// TIA Portal V15.1 export
// export: Created 2024-05-17T05:38:59.5834556Z, ExportSetting WithDefaults, DisplayName Totally Integrated Automation Portal, DisplayVersion V15.1 Update 5, DisplayName TIA Portal Openness, DisplayVersion V15.1 Update 5, DisplayName SINAMICS Startdrive Advanced, DisplayVersion V15.1, DisplayName G130, G150, S120, S150, SINAMICS MV, S210, DisplayVersion V15.1, DisplayName G110M, G120, G120C, G120D, G120P, DisplayVersion V15.1, DisplayName STEP 7 Professional, DisplayVersion V15.1 Update 5, DisplayName STEP 7 Safety, DisplayVersion V15.1, DisplayName WinCC Professional, DisplayVersion V15.1 Update 5, DisplayName SIMATIC Visualization Architect, DisplayVersion V15.1
FUNCTION "209000NCP01PNIODiag" : Void   // FC270, FBD
TITLE = 209000NCP01PNIODiag
{ S7_Optimized_Access := 'FALSE' }
AUTHOR : JS
NAME : Mot001
VERSION : 0.1
// stored: AutoNumber false, IsIECCheckEnabled false, SetENOAutomatically False, UDAEnableTagReadback false
   VAR_OUTPUT
      O_AlarmA : Bool;   // Alarm A
      O_AlarmB : Bool;   // Alarm B
      O_AlarmC : Bool;   // Alarm C
      O_AlarmD : Bool;   // Alarm D
      O_AlarmABCondition : Bool;   // Alarms resetable
      H_IAnim : Word;   // Animation bits to Icon in WinCC
   END_VAR
   VAR_TEMP   // added for the SCL form of the ladder/FBD networks
      _w1 : Bool;
   END_VAR
BEGIN

REGION Network 1: **** 1 - Inputs **** HMI Cmd
   // Extract HMI Cmd
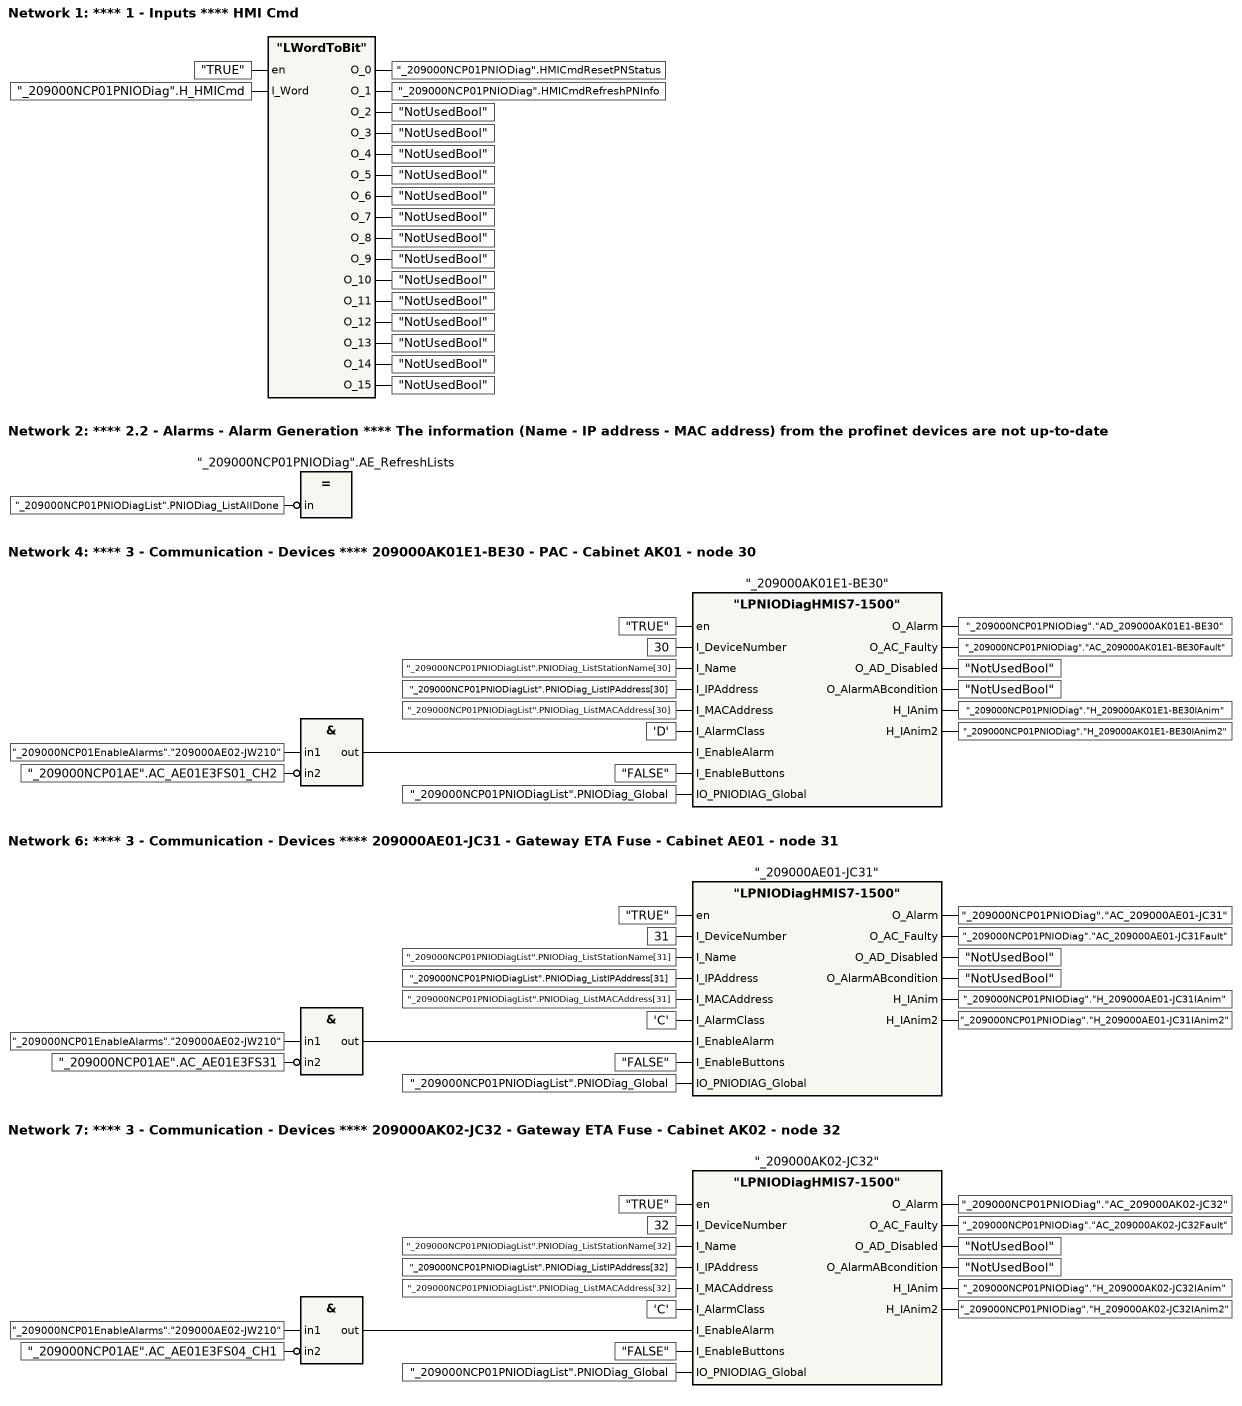
   IF "TRUE" THEN
       "LWordToBit"(I_Word := "_209000NCP01PNIODiag".H_HMICmd,
                    O_0 => "_209000NCP01PNIODiag".HMICmdResetPNStatus,
                    O_1 => "_209000NCP01PNIODiag".HMICmdRefreshPNInfo,
                    O_2 => "NotUsedBool",
                    O_3 => "NotUsedBool",
                    O_4 => "NotUsedBool",
                    O_5 => "NotUsedBool",
                    O_6 => "NotUsedBool",
                    O_7 => "NotUsedBool",
                    O_8 => "NotUsedBool",
                    O_9 => "NotUsedBool",
                    O_10 => "NotUsedBool",
                    O_11 => "NotUsedBool",
                    O_12 => "NotUsedBool",
                    O_13 => "NotUsedBool",
                    O_14 => "NotUsedBool",
                    O_15 => "NotUsedBool");
   END_IF;
END_REGION

REGION Network 2: **** 2.2 - Alarms - Alarm Generation **** The information (Name - IP address - MAC address) from the profinet devices are not up-to-date
   // The information (Name - IP address - MAC address) from the profinet devices are not up-to-date
   "_209000NCP01PNIODiag".AE_RefreshLists := NOT "_209000NCP01PNIODiagList".PNIODiag_ListAllDone;
END_REGION

REGION Network 3: **** --------------------- PAC --------------------- ****
END_REGION

REGION Network 4: **** 3 - Communication - Devices **** 209000AK01E1-BE30 - PAC - Cabinet AK01 - node 30
   // Profinet device don't exist - PAC - Cabinet AK01 - node 30
   IF "TRUE" THEN
       "_209000AK01E1-BE30"(I_DeviceNumber := 30,   // "LPNIODiagHMIS7-1500"
                            I_Name := "_209000NCP01PNIODiagList".PNIODiag_ListStationName[30],
                            I_IPAddress := "_209000NCP01PNIODiagList".PNIODiag_ListIPAddress[30],
                            I_MACAddress := "_209000NCP01PNIODiagList".PNIODiag_ListMACAddress[30],
                            I_AlarmClass := 'D',
                            I_EnableAlarm := "_209000NCP01EnableAlarms"."209000AE02-JW210" AND NOT "_209000NCP01AE".AC_AE01E3FS01_CH2,
                            I_EnableButtons := "FALSE",
                            IO_PNIODIAG_Global := "_209000NCP01PNIODiagList".PNIODiag_Global,
                            O_Alarm => "_209000NCP01PNIODiag"."AD_209000AK01E1-BE30",
                            O_AC_Faulty => "_209000NCP01PNIODiag"."AC_209000AK01E1-BE30Fault",
                            O_AD_Disabled => "NotUsedBool",
                            O_AlarmABcondition => "NotUsedBool",
                            H_IAnim => "_209000NCP01PNIODiag"."H_209000AK01E1-BE30IAnim",
                            H_IAnim2 => "_209000NCP01PNIODiag"."H_209000AK01E1-BE30IAnim2");
   END_IF;
END_REGION

REGION Network 5: **** --------------------- Gateway --------------------- ****
END_REGION

REGION Network 6: **** 3 - Communication - Devices **** 209000AE01-JC31 - Gateway ETA Fuse - Cabinet AE01 - node 31
   // Profinet device don't exist - Gateway ETA Fuse - Cabinet AE01 - node 31
   IF "TRUE" THEN
       "_209000AE01-JC31"(I_DeviceNumber := 31,   // "LPNIODiagHMIS7-1500"
                          I_Name := "_209000NCP01PNIODiagList".PNIODiag_ListStationName[31],
                          I_IPAddress := "_209000NCP01PNIODiagList".PNIODiag_ListIPAddress[31],
                          I_MACAddress := "_209000NCP01PNIODiagList".PNIODiag_ListMACAddress[31],
                          I_AlarmClass := 'C',
                          I_EnableAlarm := "_209000NCP01EnableAlarms"."209000AE02-JW210" AND NOT "_209000NCP01AE".AC_AE01E3FS31,
                          I_EnableButtons := "FALSE",
                          IO_PNIODIAG_Global := "_209000NCP01PNIODiagList".PNIODiag_Global,
                          O_Alarm => "_209000NCP01PNIODiag"."AC_209000AE01-JC31",
                          O_AC_Faulty => "_209000NCP01PNIODiag"."AC_209000AE01-JC31Fault",
                          O_AD_Disabled => "NotUsedBool",
                          O_AlarmABcondition => "NotUsedBool",
                          H_IAnim => "_209000NCP01PNIODiag"."H_209000AE01-JC31IAnim",
                          H_IAnim2 => "_209000NCP01PNIODiag"."H_209000AE01-JC31IAnim2");
   END_IF;
END_REGION

REGION Network 7: **** 3 - Communication - Devices **** 209000AK02-JC32 - Gateway ETA Fuse - Cabinet AK02 - node 32
   // Profinet device don't exist - Gateway ETA Fuse - Cabinet AK02 - node 32
   IF "TRUE" THEN
       "_209000AK02-JC32"(I_DeviceNumber := 32,   // "LPNIODiagHMIS7-1500"
                          I_Name := "_209000NCP01PNIODiagList".PNIODiag_ListStationName[32],
                          I_IPAddress := "_209000NCP01PNIODiagList".PNIODiag_ListIPAddress[32],
                          I_MACAddress := "_209000NCP01PNIODiagList".PNIODiag_ListMACAddress[32],
                          I_AlarmClass := 'C',
                          I_EnableAlarm := "_209000NCP01EnableAlarms"."209000AE02-JW210" AND NOT "_209000NCP01AE".AC_AE01E3FS04_CH1,
                          I_EnableButtons := "FALSE",
                          IO_PNIODIAG_Global := "_209000NCP01PNIODiagList".PNIODiag_Global,
                          O_Alarm => "_209000NCP01PNIODiag"."AC_209000AK02-JC32",
                          O_AC_Faulty => "_209000NCP01PNIODiag"."AC_209000AK02-JC32Fault",
                          O_AD_Disabled => "NotUsedBool",
                          O_AlarmABcondition => "NotUsedBool",
                          H_IAnim => "_209000NCP01PNIODiag"."H_209000AK02-JC32IAnim",
                          H_IAnim2 => "_209000NCP01PNIODiag"."H_209000AK02-JC32IAnim2");
   END_IF;
END_REGION

REGION Network 8: **** --------------------- ET200sp I/O --------------------- ****
END_REGION

REGION Network 9: **** 3 - Communication - Devices **** 209000AK01-JW35 - ET200sp I/O - Busnode AK01 - node 35
   // Profinet device don't exist - ET200sp I/O - Busnode AK01 - node 35
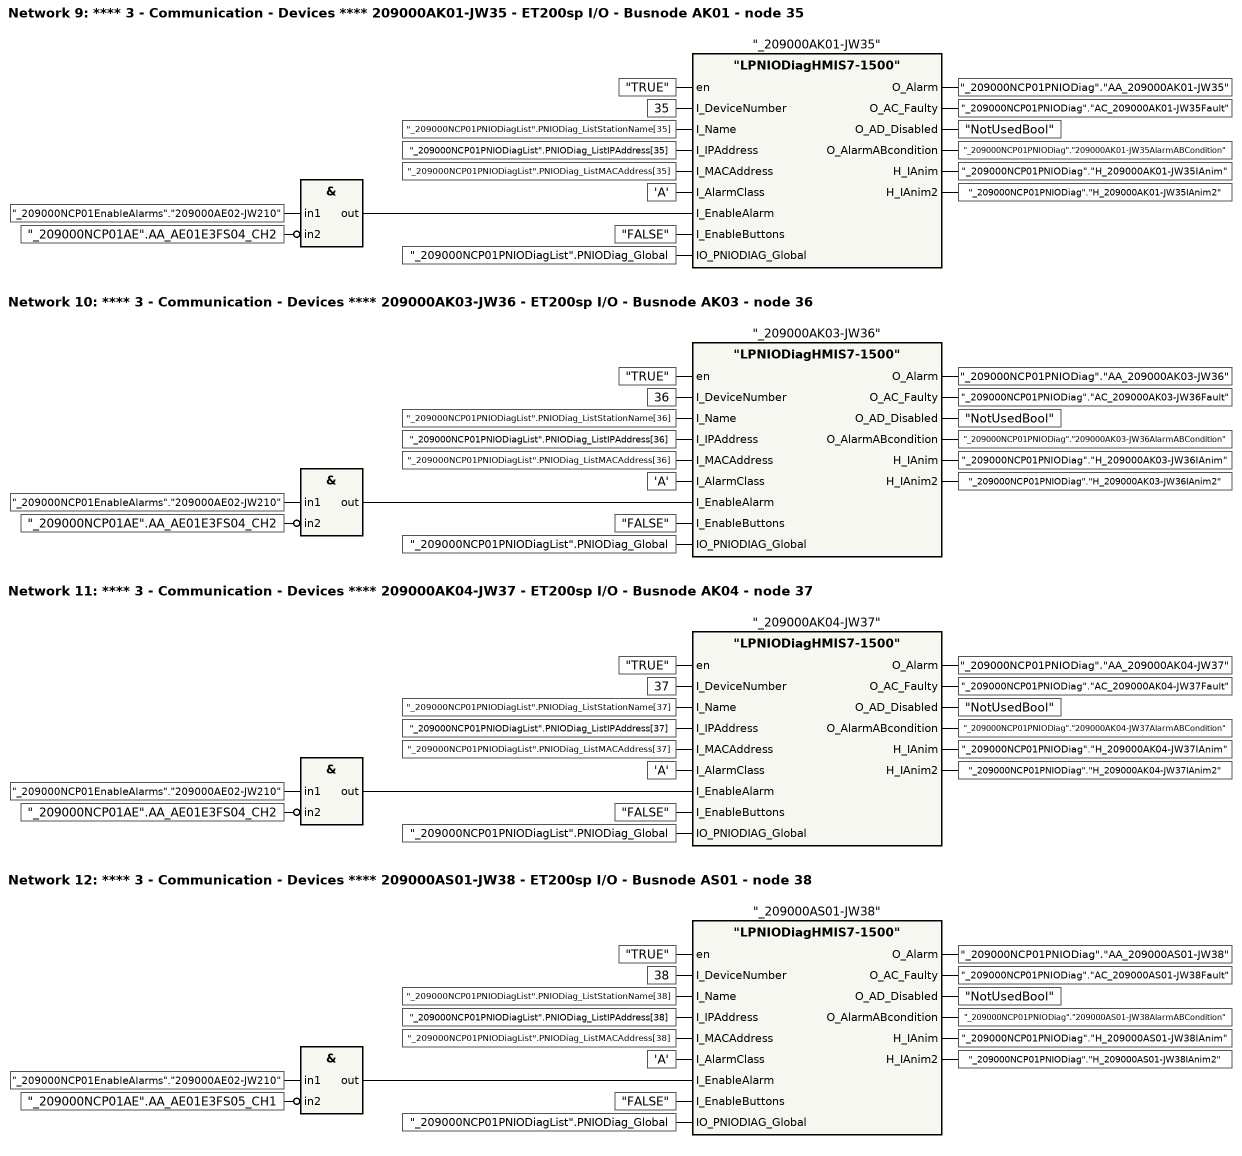
   IF "TRUE" THEN
       "_209000AK01-JW35"(I_DeviceNumber := 35,   // "LPNIODiagHMIS7-1500"
                          I_Name := "_209000NCP01PNIODiagList".PNIODiag_ListStationName[35],
                          I_IPAddress := "_209000NCP01PNIODiagList".PNIODiag_ListIPAddress[35],
                          I_MACAddress := "_209000NCP01PNIODiagList".PNIODiag_ListMACAddress[35],
                          I_AlarmClass := 'A',
                          I_EnableAlarm := "_209000NCP01EnableAlarms"."209000AE02-JW210" AND NOT "_209000NCP01AE".AA_AE01E3FS04_CH2,
                          I_EnableButtons := "FALSE",
                          IO_PNIODIAG_Global := "_209000NCP01PNIODiagList".PNIODiag_Global,
                          O_Alarm => "_209000NCP01PNIODiag"."AA_209000AK01-JW35",
                          O_AC_Faulty => "_209000NCP01PNIODiag"."AC_209000AK01-JW35Fault",
                          O_AD_Disabled => "NotUsedBool",
                          O_AlarmABcondition => "_209000NCP01PNIODiag"."209000AK01-JW35AlarmABCondition",
                          H_IAnim => "_209000NCP01PNIODiag"."H_209000AK01-JW35IAnim",
                          H_IAnim2 => "_209000NCP01PNIODiag"."H_209000AK01-JW35IAnim2");
   END_IF;
END_REGION

REGION Network 10: **** 3 - Communication - Devices **** 209000AK03-JW36 - ET200sp I/O - Busnode AK03 - node 36
   // Profinet device don't exist - ET200sp I/O - Busnode AK03 - node 36
   IF "TRUE" THEN
       "_209000AK03-JW36"(I_DeviceNumber := 36,   // "LPNIODiagHMIS7-1500"
                          I_Name := "_209000NCP01PNIODiagList".PNIODiag_ListStationName[36],
                          I_IPAddress := "_209000NCP01PNIODiagList".PNIODiag_ListIPAddress[36],
                          I_MACAddress := "_209000NCP01PNIODiagList".PNIODiag_ListMACAddress[36],
                          I_AlarmClass := 'A',
                          I_EnableAlarm := "_209000NCP01EnableAlarms"."209000AE02-JW210" AND NOT "_209000NCP01AE".AA_AE01E3FS04_CH2,
                          I_EnableButtons := "FALSE",
                          IO_PNIODIAG_Global := "_209000NCP01PNIODiagList".PNIODiag_Global,
                          O_Alarm => "_209000NCP01PNIODiag"."AA_209000AK03-JW36",
                          O_AC_Faulty => "_209000NCP01PNIODiag"."AC_209000AK03-JW36Fault",
                          O_AD_Disabled => "NotUsedBool",
                          O_AlarmABcondition => "_209000NCP01PNIODiag"."209000AK03-JW36AlarmABCondition",
                          H_IAnim => "_209000NCP01PNIODiag"."H_209000AK03-JW36IAnim",
                          H_IAnim2 => "_209000NCP01PNIODiag"."H_209000AK03-JW36IAnim2");
   END_IF;
END_REGION

REGION Network 11: **** 3 - Communication - Devices **** 209000AK04-JW37 - ET200sp I/O - Busnode AK04 - node 37
   // Profinet device don't exist - ET200sp I/O - Busnode AK04 - node 37
   IF "TRUE" THEN
       "_209000AK04-JW37"(I_DeviceNumber := 37,   // "LPNIODiagHMIS7-1500"
                          I_Name := "_209000NCP01PNIODiagList".PNIODiag_ListStationName[37],
                          I_IPAddress := "_209000NCP01PNIODiagList".PNIODiag_ListIPAddress[37],
                          I_MACAddress := "_209000NCP01PNIODiagList".PNIODiag_ListMACAddress[37],
                          I_AlarmClass := 'A',
                          I_EnableAlarm := "_209000NCP01EnableAlarms"."209000AE02-JW210" AND NOT "_209000NCP01AE".AA_AE01E3FS04_CH2,
                          I_EnableButtons := "FALSE",
                          IO_PNIODIAG_Global := "_209000NCP01PNIODiagList".PNIODiag_Global,
                          O_Alarm => "_209000NCP01PNIODiag"."AA_209000AK04-JW37",
                          O_AC_Faulty => "_209000NCP01PNIODiag"."AC_209000AK04-JW37Fault",
                          O_AD_Disabled => "NotUsedBool",
                          O_AlarmABcondition => "_209000NCP01PNIODiag"."209000AK04-JW37AlarmABCondition",
                          H_IAnim => "_209000NCP01PNIODiag"."H_209000AK04-JW37IAnim",
                          H_IAnim2 => "_209000NCP01PNIODiag"."H_209000AK04-JW37IAnim2");
   END_IF;
END_REGION

REGION Network 12: **** 3 - Communication - Devices **** 209000AS01-JW38 - ET200sp I/O - Busnode AS01 - node 38
   // Profinet device don't exist - ET200sp I/O - Busnode AS01 - node 38
   IF "TRUE" THEN
       "_209000AS01-JW38"(I_DeviceNumber := 38,   // "LPNIODiagHMIS7-1500"
                          I_Name := "_209000NCP01PNIODiagList".PNIODiag_ListStationName[38],
                          I_IPAddress := "_209000NCP01PNIODiagList".PNIODiag_ListIPAddress[38],
                          I_MACAddress := "_209000NCP01PNIODiagList".PNIODiag_ListMACAddress[38],
                          I_AlarmClass := 'A',
                          I_EnableAlarm := "_209000NCP01EnableAlarms"."209000AE02-JW210" AND NOT "_209000NCP01AE".AA_AE01E3FS05_CH1,
                          I_EnableButtons := "FALSE",
                          IO_PNIODIAG_Global := "_209000NCP01PNIODiagList".PNIODiag_Global,
                          O_Alarm => "_209000NCP01PNIODiag"."AA_209000AS01-JW38",
                          O_AC_Faulty => "_209000NCP01PNIODiag"."AC_209000AS01-JW38Fault",
                          O_AD_Disabled => "NotUsedBool",
                          O_AlarmABcondition => "_209000NCP01PNIODiag"."209000AS01-JW38AlarmABCondition",
                          H_IAnim => "_209000NCP01PNIODiag"."H_209000AS01-JW38IAnim",
                          H_IAnim2 => "_209000NCP01PNIODiag"."H_209000AS01-JW38IAnim2");
   END_IF;
END_REGION

REGION Network 13: **** 3 - Communication - Devices **** 209000AS02-JW39 - ET200sp I/O - Busnode AS02 - node 39
   // Profinet device don't exist - ET200sp I/O - Busnode AS02 - node 39
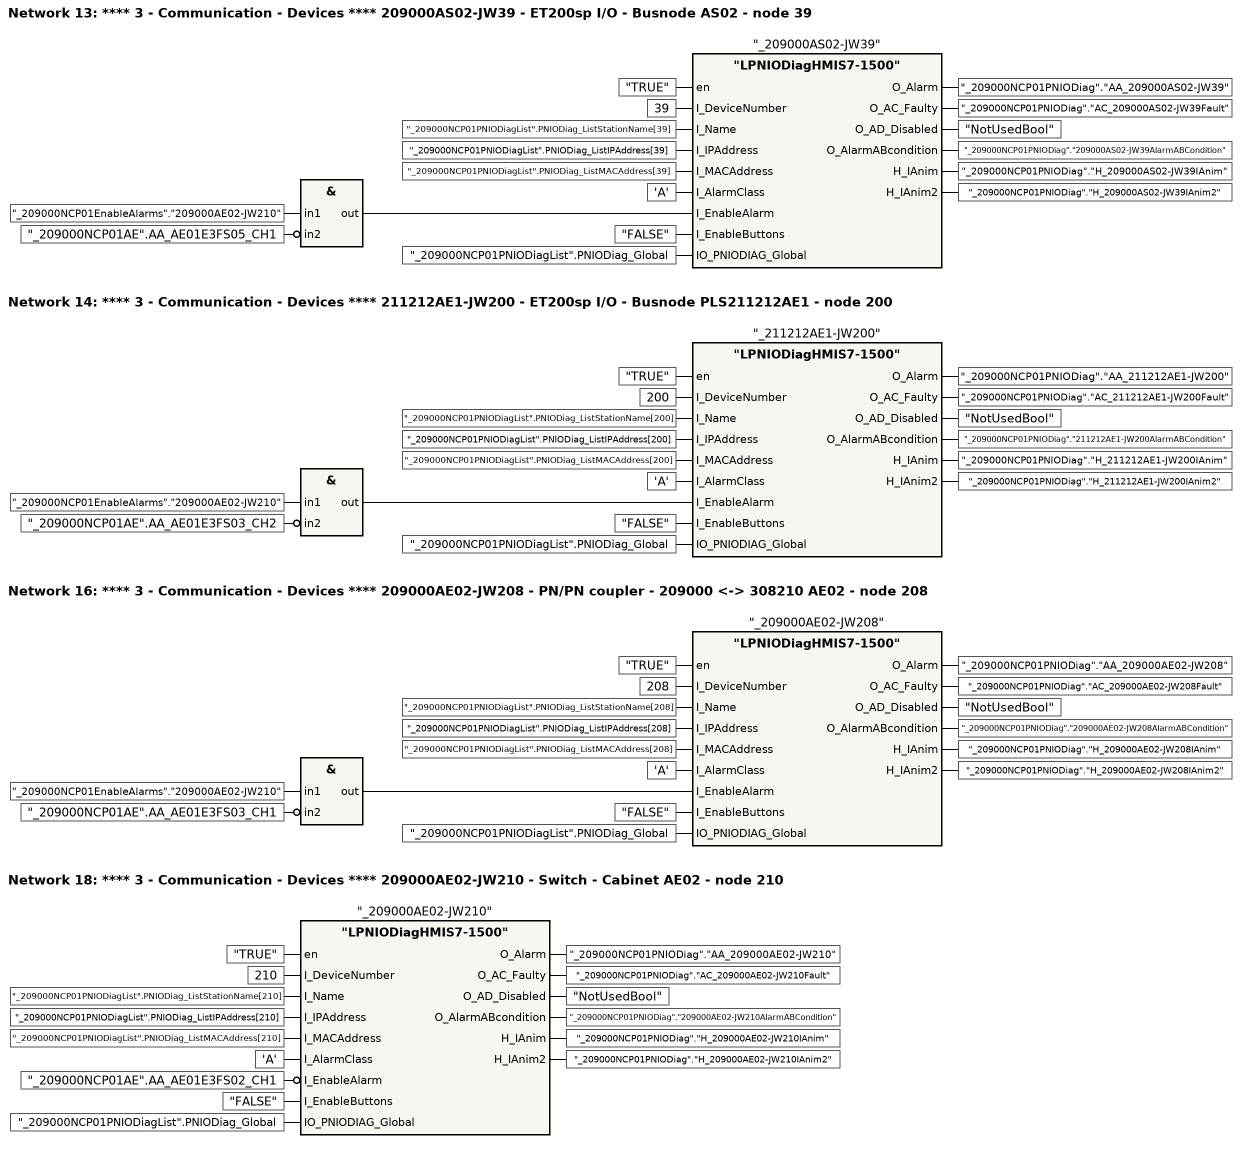
   IF "TRUE" THEN
       "_209000AS02-JW39"(I_DeviceNumber := 39,   // "LPNIODiagHMIS7-1500"
                          I_Name := "_209000NCP01PNIODiagList".PNIODiag_ListStationName[39],
                          I_IPAddress := "_209000NCP01PNIODiagList".PNIODiag_ListIPAddress[39],
                          I_MACAddress := "_209000NCP01PNIODiagList".PNIODiag_ListMACAddress[39],
                          I_AlarmClass := 'A',
                          I_EnableAlarm := "_209000NCP01EnableAlarms"."209000AE02-JW210" AND NOT "_209000NCP01AE".AA_AE01E3FS05_CH1,
                          I_EnableButtons := "FALSE",
                          IO_PNIODIAG_Global := "_209000NCP01PNIODiagList".PNIODiag_Global,
                          O_Alarm => "_209000NCP01PNIODiag"."AA_209000AS02-JW39",
                          O_AC_Faulty => "_209000NCP01PNIODiag"."AC_209000AS02-JW39Fault",
                          O_AD_Disabled => "NotUsedBool",
                          O_AlarmABcondition => "_209000NCP01PNIODiag"."209000AS02-JW39AlarmABCondition",
                          H_IAnim => "_209000NCP01PNIODiag"."H_209000AS02-JW39IAnim",
                          H_IAnim2 => "_209000NCP01PNIODiag"."H_209000AS02-JW39IAnim2");
   END_IF;
END_REGION

REGION Network 14: **** 3 - Communication - Devices **** 211212AE1-JW200 - ET200sp I/O - Busnode PLS211212AE1 - node 200
   // Profinet device don't exist - ET200sp I/O - Busnode PLS211212AE1 - node 200
   IF "TRUE" THEN
       "_211212AE1-JW200"(I_DeviceNumber := 200,   // "LPNIODiagHMIS7-1500"
                          I_Name := "_209000NCP01PNIODiagList".PNIODiag_ListStationName[200],
                          I_IPAddress := "_209000NCP01PNIODiagList".PNIODiag_ListIPAddress[200],
                          I_MACAddress := "_209000NCP01PNIODiagList".PNIODiag_ListMACAddress[200],
                          I_AlarmClass := 'A',
                          I_EnableAlarm := "_209000NCP01EnableAlarms"."209000AE02-JW210" AND NOT "_209000NCP01AE".AA_AE01E3FS03_CH2,
                          I_EnableButtons := "FALSE",
                          IO_PNIODIAG_Global := "_209000NCP01PNIODiagList".PNIODiag_Global,
                          O_Alarm => "_209000NCP01PNIODiag"."AA_211212AE1-JW200",
                          O_AC_Faulty => "_209000NCP01PNIODiag"."AC_211212AE1-JW200Fault",
                          O_AD_Disabled => "NotUsedBool",
                          O_AlarmABcondition => "_209000NCP01PNIODiag"."211212AE1-JW200AlarmABCondition",
                          H_IAnim => "_209000NCP01PNIODiag"."H_211212AE1-JW200IAnim",
                          H_IAnim2 => "_209000NCP01PNIODiag"."H_211212AE1-JW200IAnim2");
   END_IF;
END_REGION

REGION Network 15: **** --------------------- PN/PN coupler --------------------- ****
END_REGION

REGION Network 16: **** 3 - Communication - Devices **** 209000AE02-JW208 - PN/PN coupler - 209000 <-> 308210 AE02 - node 208
   // Profinet device don't exist - PN/PN coupler - 209000 <-> 308210 AE02 - node 208
   IF "TRUE" THEN
       "_209000AE02-JW208"(I_DeviceNumber := 208,   // "LPNIODiagHMIS7-1500"
                           I_Name := "_209000NCP01PNIODiagList".PNIODiag_ListStationName[208],
                           I_IPAddress := "_209000NCP01PNIODiagList".PNIODiag_ListIPAddress[208],
                           I_MACAddress := "_209000NCP01PNIODiagList".PNIODiag_ListMACAddress[208],
                           I_AlarmClass := 'A',
                           I_EnableAlarm := "_209000NCP01EnableAlarms"."209000AE02-JW210" AND NOT "_209000NCP01AE".AA_AE01E3FS03_CH1,
                           I_EnableButtons := "FALSE",
                           IO_PNIODIAG_Global := "_209000NCP01PNIODiagList".PNIODiag_Global,
                           O_Alarm => "_209000NCP01PNIODiag"."AA_209000AE02-JW208",
                           O_AC_Faulty => "_209000NCP01PNIODiag"."AC_209000AE02-JW208Fault",
                           O_AD_Disabled => "NotUsedBool",
                           O_AlarmABcondition => "_209000NCP01PNIODiag"."209000AE02-JW208AlarmABCondition",
                           H_IAnim => "_209000NCP01PNIODiag"."H_209000AE02-JW208IAnim",
                           H_IAnim2 => "_209000NCP01PNIODiag"."H_209000AE02-JW208IAnim2");
   END_IF;
END_REGION

REGION Network 17: **** --------------------- Switch --------------------- ****
END_REGION

REGION Network 18: **** 3 - Communication - Devices **** 209000AE02-JW210 - Switch - Cabinet AE02 - node 210
   // Profinet device don't exist - Switch - Cabinet AE02 - node 210
   IF "TRUE" THEN
       "_209000AE02-JW210"(I_DeviceNumber := 210,   // "LPNIODiagHMIS7-1500"
                           I_Name := "_209000NCP01PNIODiagList".PNIODiag_ListStationName[210],
                           I_IPAddress := "_209000NCP01PNIODiagList".PNIODiag_ListIPAddress[210],
                           I_MACAddress := "_209000NCP01PNIODiagList".PNIODiag_ListMACAddress[210],
                           I_AlarmClass := 'A',
                           I_EnableAlarm := NOT "_209000NCP01AE".AA_AE01E3FS02_CH1,
                           I_EnableButtons := "FALSE",
                           IO_PNIODIAG_Global := "_209000NCP01PNIODiagList".PNIODiag_Global,
                           O_Alarm => "_209000NCP01PNIODiag"."AA_209000AE02-JW210",
                           O_AC_Faulty => "_209000NCP01PNIODiag"."AC_209000AE02-JW210Fault",
                           O_AD_Disabled => "NotUsedBool",
                           O_AlarmABcondition => "_209000NCP01PNIODiag"."209000AE02-JW210AlarmABCondition",
                           H_IAnim => "_209000NCP01PNIODiag"."H_209000AE02-JW210IAnim",
                           H_IAnim2 => "_209000NCP01PNIODiag"."H_209000AE02-JW210IAnim2");
   END_IF;
END_REGION

REGION Network 19: **** 3 - Communication - Devices **** 209000AE02-JW211 - Switch - Cabinet AE02 - node 211
   // Profinet device don't exist - Switch - Cabinet AE02 - node 211
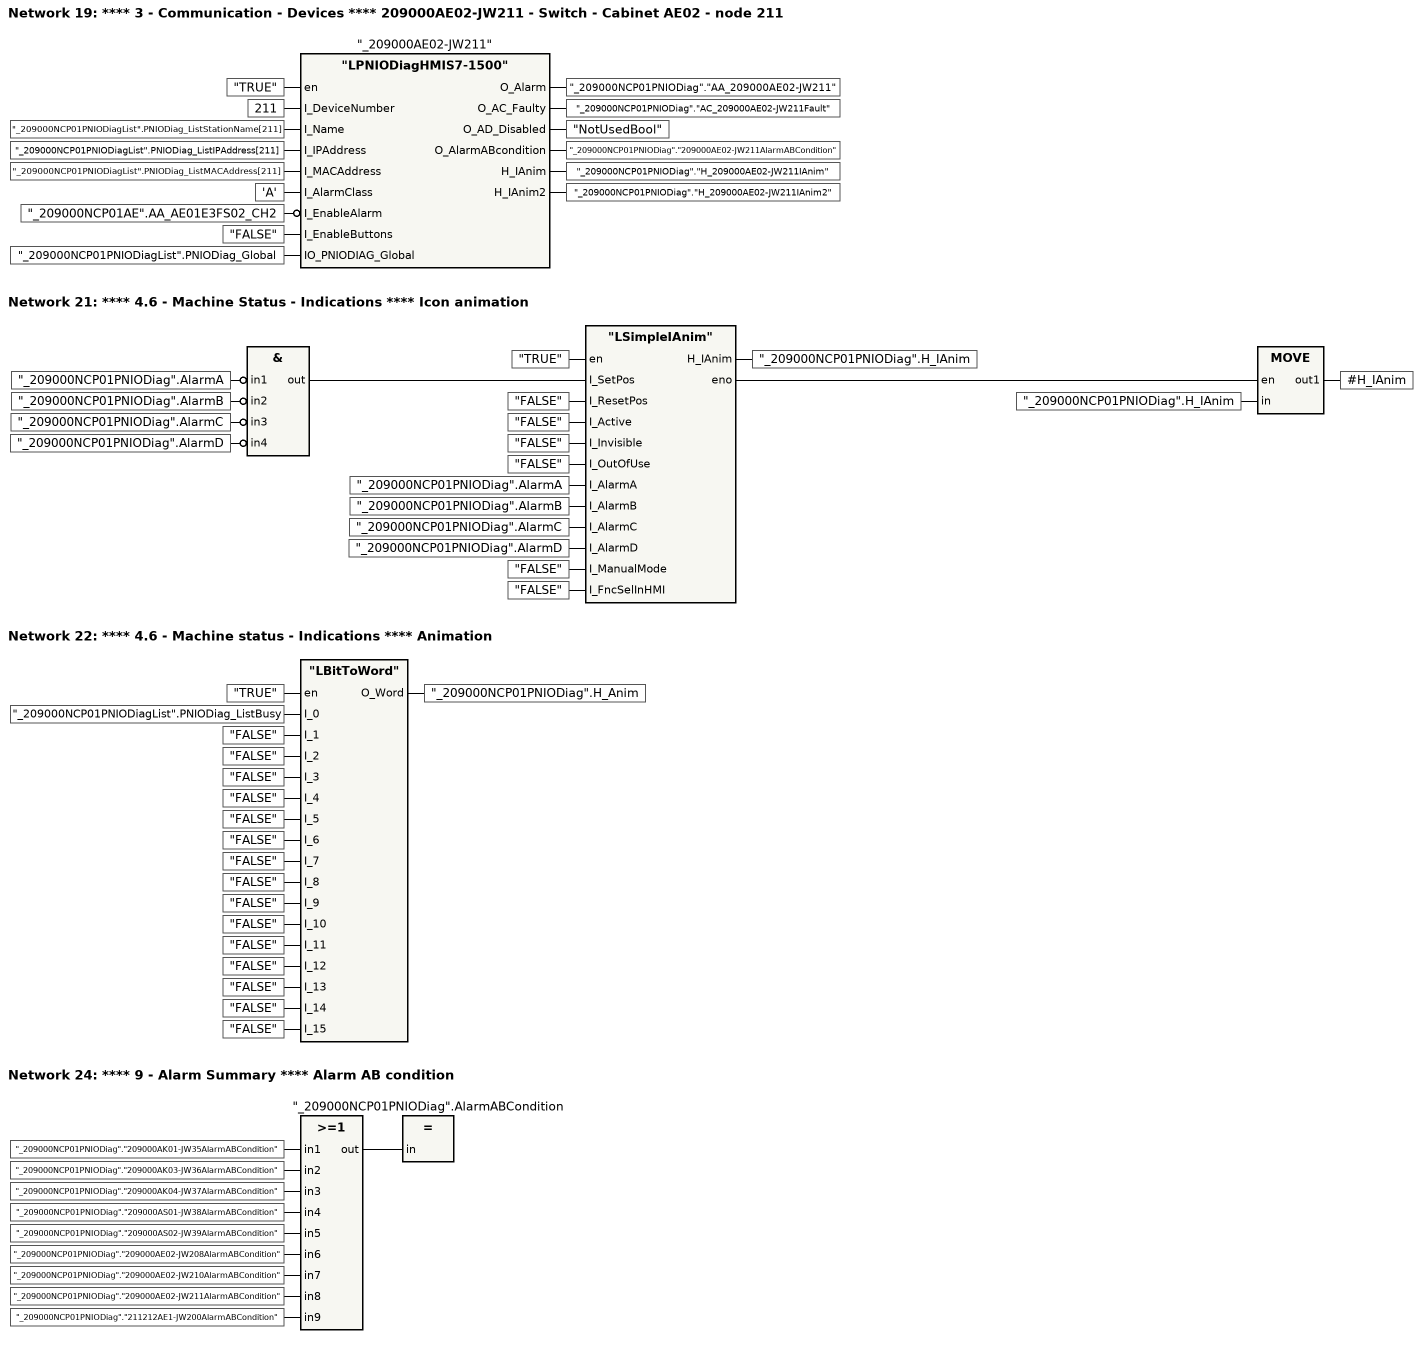
   IF "TRUE" THEN
       "_209000AE02-JW211"(I_DeviceNumber := 211,   // "LPNIODiagHMIS7-1500"
                           I_Name := "_209000NCP01PNIODiagList".PNIODiag_ListStationName[211],
                           I_IPAddress := "_209000NCP01PNIODiagList".PNIODiag_ListIPAddress[211],
                           I_MACAddress := "_209000NCP01PNIODiagList".PNIODiag_ListMACAddress[211],
                           I_AlarmClass := 'A',
                           I_EnableAlarm := NOT "_209000NCP01AE".AA_AE01E3FS02_CH2,
                           I_EnableButtons := "FALSE",
                           IO_PNIODIAG_Global := "_209000NCP01PNIODiagList".PNIODiag_Global,
                           O_Alarm => "_209000NCP01PNIODiag"."AA_209000AE02-JW211",
                           O_AC_Faulty => "_209000NCP01PNIODiag"."AC_209000AE02-JW211Fault",
                           O_AD_Disabled => "NotUsedBool",
                           O_AlarmABcondition => "_209000NCP01PNIODiag"."209000AE02-JW211AlarmABCondition",
                           H_IAnim => "_209000NCP01PNIODiag"."H_209000AE02-JW211IAnim",
                           H_IAnim2 => "_209000NCP01PNIODiag"."H_209000AE02-JW211IAnim2");
   END_IF;
END_REGION

REGION Network 20: **** -------------------------------------------------- ****
END_REGION

REGION Network 21: **** 4.6 - Machine Status - Indications **** Icon animation
   // Icon animation
   "LSimpleIAnim"(EN := "TRUE",
                  I_SetPos := NOT "_209000NCP01PNIODiag".AlarmA AND NOT "_209000NCP01PNIODiag".AlarmB AND NOT "_209000NCP01PNIODiag".AlarmC AND NOT "_209000NCP01PNIODiag".AlarmD,
                  I_ResetPos := "FALSE",
                  I_Active := "FALSE",
                  I_Invisible := "FALSE",
                  I_OutOfUse := "FALSE",
                  I_AlarmA := "_209000NCP01PNIODiag".AlarmA,
                  I_AlarmB := "_209000NCP01PNIODiag".AlarmB,
                  I_AlarmC := "_209000NCP01PNIODiag".AlarmC,
                  I_AlarmD := "_209000NCP01PNIODiag".AlarmD,
                  I_ManualMode := "FALSE",
                  I_FncSelInHMI := "FALSE",
                  H_IAnim => "_209000NCP01PNIODiag".H_IAnim,
                  ENO => #_w1);
   IF #_w1 THEN #H_IAnim := "_209000NCP01PNIODiag".H_IAnim; END_IF;
END_REGION

REGION Network 22: **** 4.6 - Machine status - Indications **** Animation
   // Animation
   IF "TRUE" THEN
       "LBitToWord"(I_0 := "_209000NCP01PNIODiagList".PNIODiag_ListBusy,
                    I_1 := "FALSE",
                    I_2 := "FALSE",
                    I_3 := "FALSE",
                    I_4 := "FALSE",
                    I_5 := "FALSE",
                    I_6 := "FALSE",
                    I_7 := "FALSE",
                    I_8 := "FALSE",
                    I_9 := "FALSE",
                    I_10 := "FALSE",
                    I_11 := "FALSE",
                    I_12 := "FALSE",
                    I_13 := "FALSE",
                    I_14 := "FALSE",
                    I_15 := "FALSE",
                    O_Word => "_209000NCP01PNIODiag".H_Anim);
   END_IF;
END_REGION

NETWORK
TITLE = **** 4.6 - Machine Status - Indications **** Animation DB number
// DB number
      OPN   "_209000NCP01PNIODiag";
      L     DBNO;
      T     "_209000NCP01PNIODiag".H_DBnr;

REGION Network 24: **** 9 - Alarm Summary **** Alarm AB condition
   // Summary of Alarm AB condition
   "_209000NCP01PNIODiag".AlarmABCondition := "_209000NCP01PNIODiag"."209000AK01-JW35AlarmABCondition" OR "_209000NCP01PNIODiag"."209000AK03-JW36AlarmABCondition" OR "_209000NCP01PNIODiag"."209000AK04-JW37AlarmABCondition" OR "_209000NCP01PNIODiag"."209000AS01-JW38AlarmABCondition" OR "_209000NCP01PNIODiag"."209000AS02-JW39AlarmABCondition" OR "_209000NCP01PNIODiag"."209000AE02-JW208AlarmABCondition" OR "_209000NCP01PNIODiag"."209000AE02-JW210AlarmABCondition" OR "_209000NCP01PNIODiag"."209000AE02-JW211AlarmABCondition" OR "_209000NCP01PNIODiag"."211212AE1-JW200AlarmABCondition";
END_REGION

REGION Network 25: **** 9 - Alarm Summary **** Alarm A
   // Summary of alarms A
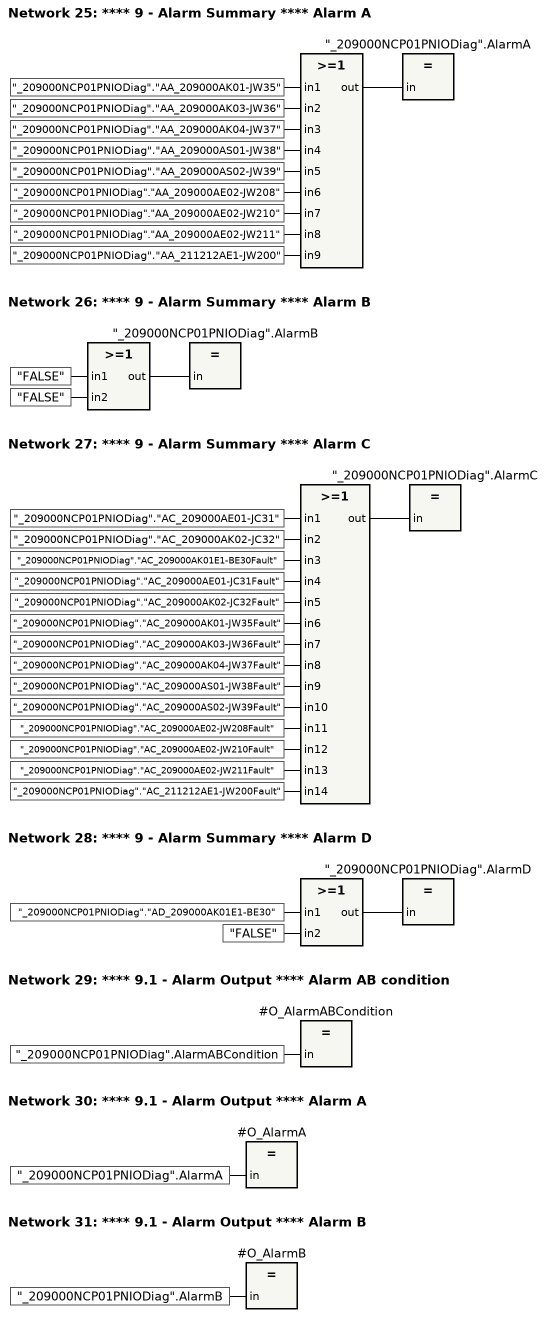
   "_209000NCP01PNIODiag".AlarmA := "_209000NCP01PNIODiag"."AA_209000AK01-JW35" OR "_209000NCP01PNIODiag"."AA_209000AK03-JW36" OR "_209000NCP01PNIODiag"."AA_209000AK04-JW37" OR "_209000NCP01PNIODiag"."AA_209000AS01-JW38" OR "_209000NCP01PNIODiag"."AA_209000AS02-JW39" OR "_209000NCP01PNIODiag"."AA_209000AE02-JW208" OR "_209000NCP01PNIODiag"."AA_209000AE02-JW210" OR "_209000NCP01PNIODiag"."AA_209000AE02-JW211" OR "_209000NCP01PNIODiag"."AA_211212AE1-JW200";
END_REGION

REGION Network 26: **** 9 - Alarm Summary **** Alarm B
   // Summary of alarms B
   "_209000NCP01PNIODiag".AlarmB := "FALSE" OR "FALSE";
END_REGION

REGION Network 27: **** 9 - Alarm Summary **** Alarm C
   // Summary of alarms C
   "_209000NCP01PNIODiag".AlarmC := "_209000NCP01PNIODiag"."AC_209000AE01-JC31" OR "_209000NCP01PNIODiag"."AC_209000AK02-JC32" OR "_209000NCP01PNIODiag"."AC_209000AK01E1-BE30Fault" OR "_209000NCP01PNIODiag"."AC_209000AE01-JC31Fault" OR "_209000NCP01PNIODiag"."AC_209000AK02-JC32Fault" OR "_209000NCP01PNIODiag"."AC_209000AK01-JW35Fault" OR "_209000NCP01PNIODiag"."AC_209000AK03-JW36Fault" OR "_209000NCP01PNIODiag"."AC_209000AK04-JW37Fault" OR "_209000NCP01PNIODiag"."AC_209000AS01-JW38Fault" OR "_209000NCP01PNIODiag"."AC_209000AS02-JW39Fault" OR "_209000NCP01PNIODiag"."AC_209000AE02-JW208Fault" OR "_209000NCP01PNIODiag"."AC_209000AE02-JW210Fault" OR "_209000NCP01PNIODiag"."AC_209000AE02-JW211Fault" OR "_209000NCP01PNIODiag"."AC_211212AE1-JW200Fault";
END_REGION

REGION Network 28: **** 9 - Alarm Summary **** Alarm D
   // Summary of alarms D
   "_209000NCP01PNIODiag".AlarmD := "_209000NCP01PNIODiag"."AD_209000AK01E1-BE30" OR "FALSE";
END_REGION

REGION Network 29: **** 9.1 - Alarm Output **** Alarm AB condition
   // Alarm AB condition
   #O_AlarmABCondition := "_209000NCP01PNIODiag".AlarmABCondition;
END_REGION

REGION Network 30: **** 9.1 - Alarm Output **** Alarm A
   // Output Alarm A
   #O_AlarmA := "_209000NCP01PNIODiag".AlarmA;
END_REGION

REGION Network 31: **** 9.1 - Alarm Output **** Alarm B
   // Output Alarm B
   #O_AlarmB := "_209000NCP01PNIODiag".AlarmB;
END_REGION

REGION Network 32: **** 9.1 - Alarm Output **** Alarm C
   // Output Alarm A
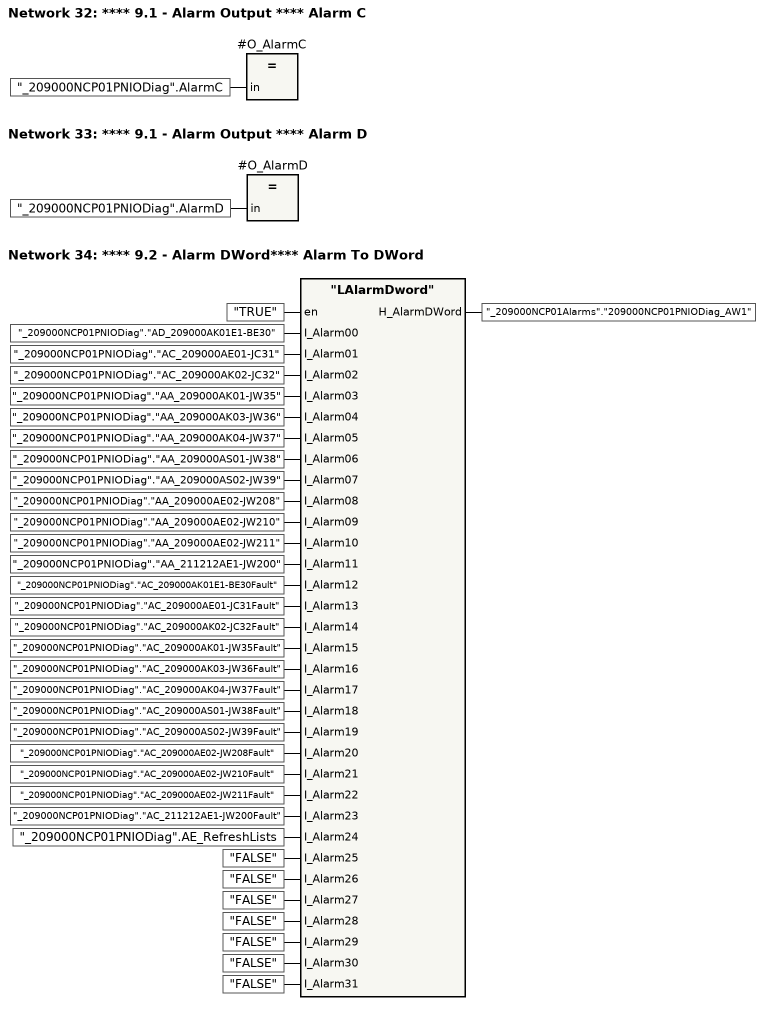
   #O_AlarmC := "_209000NCP01PNIODiag".AlarmC;
END_REGION

REGION Network 33: **** 9.1 - Alarm Output **** Alarm D
   // Output Alarm D
   #O_AlarmD := "_209000NCP01PNIODiag".AlarmD;
END_REGION

REGION Network 34: **** 9.2 - Alarm DWord**** Alarm To DWord
   // Alarm Word
   IF "TRUE" THEN
       "LAlarmDword"(I_Alarm00 := "_209000NCP01PNIODiag"."AD_209000AK01E1-BE30",
                     I_Alarm01 := "_209000NCP01PNIODiag"."AC_209000AE01-JC31",
                     I_Alarm02 := "_209000NCP01PNIODiag"."AC_209000AK02-JC32",
                     I_Alarm03 := "_209000NCP01PNIODiag"."AA_209000AK01-JW35",
                     I_Alarm04 := "_209000NCP01PNIODiag"."AA_209000AK03-JW36",
                     I_Alarm05 := "_209000NCP01PNIODiag"."AA_209000AK04-JW37",
                     I_Alarm06 := "_209000NCP01PNIODiag"."AA_209000AS01-JW38",
                     I_Alarm07 := "_209000NCP01PNIODiag"."AA_209000AS02-JW39",
                     I_Alarm08 := "_209000NCP01PNIODiag"."AA_209000AE02-JW208",
                     I_Alarm09 := "_209000NCP01PNIODiag"."AA_209000AE02-JW210",
                     I_Alarm10 := "_209000NCP01PNIODiag"."AA_209000AE02-JW211",
                     I_Alarm11 := "_209000NCP01PNIODiag"."AA_211212AE1-JW200",
                     I_Alarm12 := "_209000NCP01PNIODiag"."AC_209000AK01E1-BE30Fault",
                     I_Alarm13 := "_209000NCP01PNIODiag"."AC_209000AE01-JC31Fault",
                     I_Alarm14 := "_209000NCP01PNIODiag"."AC_209000AK02-JC32Fault",
                     I_Alarm15 := "_209000NCP01PNIODiag"."AC_209000AK01-JW35Fault",
                     I_Alarm16 := "_209000NCP01PNIODiag"."AC_209000AK03-JW36Fault",
                     I_Alarm17 := "_209000NCP01PNIODiag"."AC_209000AK04-JW37Fault",
                     I_Alarm18 := "_209000NCP01PNIODiag"."AC_209000AS01-JW38Fault",
                     I_Alarm19 := "_209000NCP01PNIODiag"."AC_209000AS02-JW39Fault",
                     I_Alarm20 := "_209000NCP01PNIODiag"."AC_209000AE02-JW208Fault",
                     I_Alarm21 := "_209000NCP01PNIODiag"."AC_209000AE02-JW210Fault",
                     I_Alarm22 := "_209000NCP01PNIODiag"."AC_209000AE02-JW211Fault",
                     I_Alarm23 := "_209000NCP01PNIODiag"."AC_211212AE1-JW200Fault",
                     I_Alarm24 := "_209000NCP01PNIODiag".AE_RefreshLists,
                     I_Alarm25 := "FALSE",
                     I_Alarm26 := "FALSE",
                     I_Alarm27 := "FALSE",
                     I_Alarm28 := "FALSE",
                     I_Alarm29 := "FALSE",
                     I_Alarm30 := "FALSE",
                     I_Alarm31 := "FALSE",
                     H_AlarmDWord => "_209000NCP01Alarms"."209000NCP01PNIODiag_AW1");
   END_IF;
END_REGION
END_FUNCTION
